FUNCTION_BLOCK fbAssignBadBstCtrl
VAR_INPUT

	bMain			: BOOL;
	bAutoStart		: BOOL;
	bBasketCFM		: BOOL;

	bAssignBit1		: BOOL;
	bAssignBit2		: BOOL;
	bAssignBit3		: BOOL;
	bAssignBit4		: BOOL;
	bAssignBit5		: BOOL;
	bAssignBit6		: BOOL;
	bAssignBit7		: BOOL;
	bAssignBit8		: BOOL;
	bAssignBit9		: BOOL;
	bAssignBit10		: BOOL;
	bAssignBit11		: BOOL;
	bAssignBit12		: BOOL;
	bAssignBit13		: BOOL;
	bAssignBit14		: BOOL;
	bAssignBit15		: BOOL;
	bAssignBit16		: BOOL;
	bAssignBit17		: BOOL;
	bAssignBit18		: BOOL;
	bAssignBit19		: BOOL;
	bAssignBit20		: BOOL;
	bAssignBit21		: BOOL;
	bAssignBit22		: BOOL;
	bAssignBit23		: BOOL;
	bAssignBit24		: BOOL;
	bAssignBit25		: BOOL;
	bAssignBit26		: BOOL;
	bAssignBit27		: BOOL;
	bAssignBit28		: BOOL;
	bAssignBit29		: BOOL;
	bAssignBit30		: BOOL;

END_VAR
VAR_IN_OUT

	SbadBasket		: STRING(50);

END_VAR
VAR
	TRIG1: R_TRIG;
END_VAR
VAR // added by the converter: edge detectors and wires of the graphical bodies
    _w1 : ANY;
END_VAR

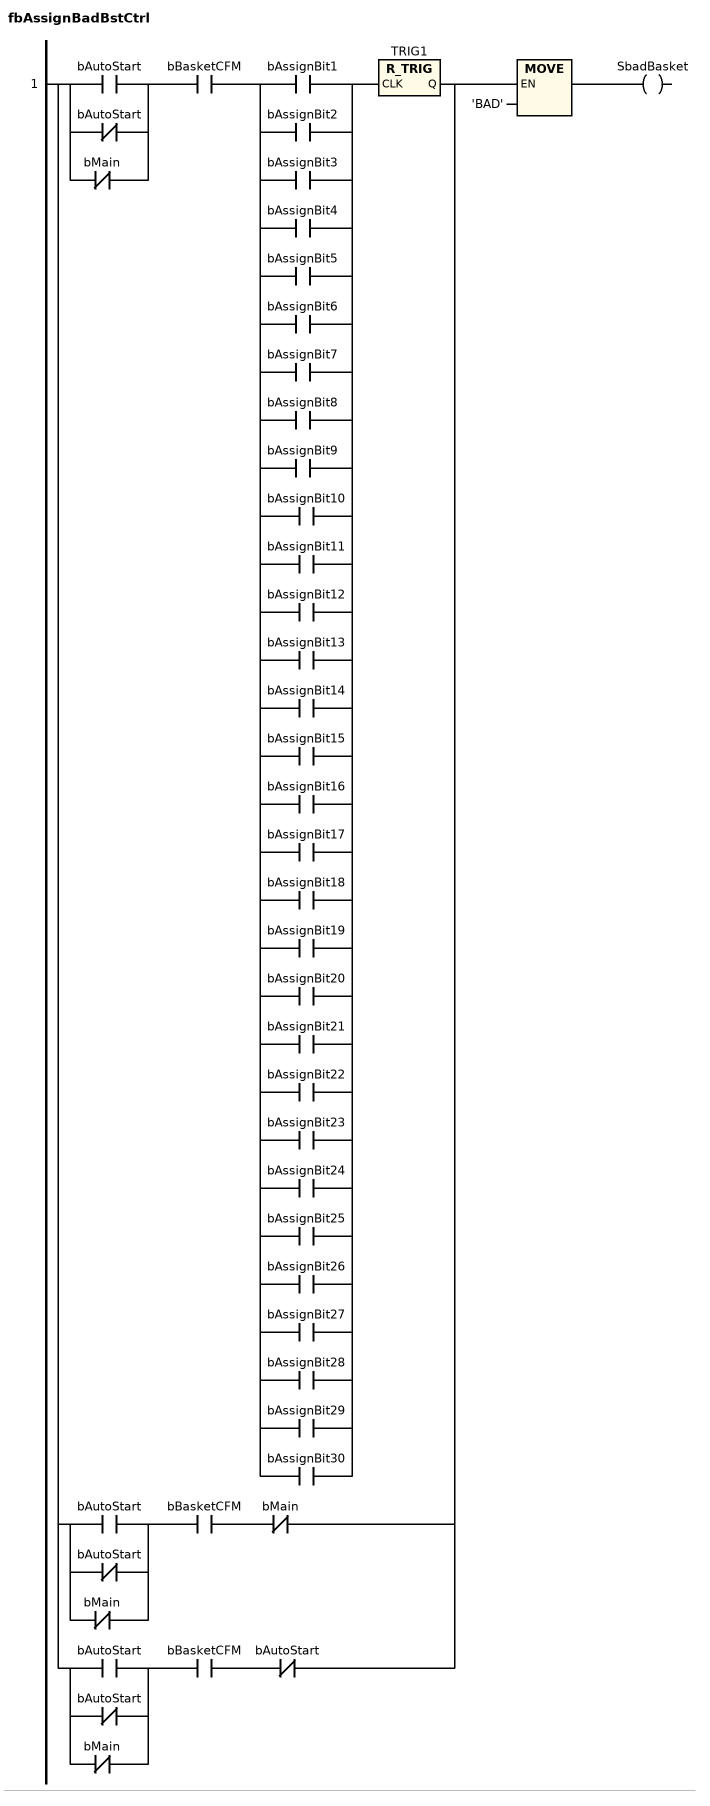
// NETWORK 1
TRIG1(CLK := ((bAutoStart OR NOT bAutoStart OR NOT bMain) AND bBasketCFM) AND (bAssignBit1 OR bAssignBit2 OR bAssignBit3 OR bAssignBit4 OR bAssignBit5 OR bAssignBit6 OR bAssignBit7 OR bAssignBit8 OR bAssignBit9 OR bAssignBit10 OR bAssignBit11 OR bAssignBit12 OR bAssignBit13 OR bAssignBit14 OR bAssignBit15 OR bAssignBit16 OR bAssignBit17 OR bAssignBit18 OR bAssignBit19 OR bAssignBit20 OR bAssignBit21 OR bAssignBit22 OR bAssignBit23 OR bAssignBit24 OR bAssignBit25 OR bAssignBit26 OR bAssignBit27 OR bAssignBit28 OR bAssignBit29 OR bAssignBit30)); // R_TRIG
IF TRIG1.Q OR ((bAutoStart OR NOT bAutoStart OR NOT bMain) AND bBasketCFM) AND NOT bMain OR ((bAutoStart OR NOT bAutoStart OR NOT bMain) AND bBasketCFM) AND NOT bAutoStart THEN
    _w1 := 'BAD';
END_IF
SbadBasket := _w1;

END_FUNCTION_BLOCK

(* stored: Version 1.1.0.1, ProductVersion 3.1.4024.12
   POU fbAssignBadBstCtrl: Id {7d18d7d3-a95f-4ba7-a30d-393fc9537329}, SpecialFunc None *)
